PROGRAM PRG_4_LOG
VAR
    fbLogHandler: FB_LogHandler;
END_VAR

fbLogHandler();

END_PROGRAM

(* stored: Version 1.1.0.1
   POU PRG_4_LOG: Id {481906ac-7b04-0833-0c94-35bab68178b7}, SpecialFunc None *)
